Universal Robots PolyScope program: path_offset_square_weave_UR10_text.urp

Program path_offset_square_weave_UR10 (installation=path_offset_square_weave_UR10 directory=/home/ask/git/polyscope/staging/programs createdIn=5.5.0.0 lastSavedIn=5.5.0.0 robotSerialNumber=20175099999)
Calibrated DH parameters: a=[0, -0.6127, -0.57155, 0, 0, 0]; d=[0.1807, 0, 0, 0.17415, 0.11985, 0.11655]; alpha=[1.570796, 0, 0, 1.570796, -1.570796, 0]; deltaTheta=[0, 0, 0, 0, 0, 0]
Robot Program (runOnlyOnce=true)
  MoveP speed 8 mm/s, acceleration 1200 mm/s^2 (blendRadius=0.025 useActiveTCP=true) feature=Base
    Waypoint start_pos: TCP in base x=-200 y=-700 z=100 mm, rx=0 ry=-3.1412 rz=0 rad; joints [-92.101, -119.704, -120.57, -29.725, 89.977, -2.101] deg; TCP offset x=0 y=0 z=0 mm, rx=0 ry=0 rz=0 rad
    Waypoint end_pos: TCP in base x=100 y=-700 z=100 mm, rx=0 ry=3.1168 rz=0 rad; joints [-67.836, -118.644, -123.011, -27.808, 91.317, 22.17] deg; TCP offset x=0 y=0 z=0 mm, rx=0 ry=0 rz=0 rad
Thread Thread_1 (runOnlyOnce=false)
  Folder setup
    ctrl_frequency := 500.0
    weave_frequency := 3.0
    amplitude := 0.006
    speed := 0.008
    in_out_distance := amplitude
    follow_distance := (speed / weave_frequency) / 2.0
    cycle_distance := (4.0 * in_out_distance) + (2.0 * follow_distance)
    in_out_duration := floor((ctrl_frequency / weave_frequency) * (in_out_distance / cycle_distance))
    follow_duration := floor((ctrl_frequency / weave_frequency) * (follow_distance / cycle_distance))
    cycle_duration := (4 * in_out_duration) + (2 * follow_duration)
    in_out_addition := in_out_distance / in_out_duration
    follow_mult := 2.0 * (in_out_duration / follow_duration)
  Folder enable
    offset := [0.0, 0.0, 0.0, 0.0, 0.0, 0.0]
    i := 0
    Script: path_offset_enable()
    alpha := 0.165
    Script: path_offset_set_alpha_filter(alpha)
  Folder weave
    Loop Forever
      traj_vel := get_target_tcp_speed_along_path()
      traj_vel_pos := [traj_vel[0], traj_vel[1], traj_vel[2]]
      If i<in_out_duration
        Script: offset[0] = offset[0]-(norm(traj_vel_pos) / ctrl_frequency)
        Script: offset[1] = offset[1]+in_out_addition
      ElseIf i<(in_out_duration+follow_duration)
        Script: offset[0] = offset[0]+(follow_mult * (norm(traj_vel_pos) / ctrl_frequency))
      ElseIf i<((3 * in_out_duration) + follow_duration)
        Script: offset[0] = offset[0]-(norm(traj_vel_pos) / ctrl_frequency)
        Script: offset[1] = offset[1]-in_out_addition
      ElseIf i<((3 * in_out_duration) + (2 * follow_duration))
        Script: offset[0] = offset[0]+(follow_mult * (norm(traj_vel_pos) / ctrl_frequency))
      Else 
        Script: offset[0] = offset[0]-(norm(traj_vel_pos) / ctrl_frequency)
        Script: offset[1] = offset[1]+in_out_addition
      Script: path_offset_set(offset, 3)
      i := i+1
      If i≥cycle_duration
        i := 0
      Script: sync()
